Fanuc KAREL source: wextindep.kl

PROGRAM wextindep
%NOLOCKGROUP
VAR
  p : POSITION
  q : POSITION
  i : INTEGER
  r : REAL
BEGIN
  WITH $EXT_INDEP = TRUE MOVE TO p
END wextindep
